FUNCTION_BLOCK NodePack_PlcBasicLiterals IMPLEMENTS I_NodePack
VAR
	nodeFactory_Literal_BOOL : NodeFactory_Literal_BOOL;
END_VAR

METHOD PUBLIC RegisterWithGraph
VAR_INPUT
	TcGraph : I_TcGraph;
END_VAR
TcGraph.RegisterNodeFactoryByType('PLC Basic/Literals/BOOL',nodeFactory_Literal_BOOL);
END_METHOD

END_FUNCTION_BLOCK

(* stored: Version 1.1.0.1, ProductVersion 3.1.4024.12
   POU NodePack_PlcBasicLiterals: Id {09b91d76-6524-009b-0de9-751b027e358a}, SpecialFunc None
   Method RegisterWithGraph: Id {3ef8db7d-47fb-090b-3597-c30640cd5056} *)
